PROGRAM Control_LD

VAR	
	Btn1_pressed: BOOL; // Either ixButtLevel1 or ixButtElevat1 was pressed
	Btn2_pressed: BOOL; // Either ixButtLevel2 or ixButtElevat2 was pressed
	Btn3_pressed: BOOL; // Either ixButtLevel3 or ixButtElevat3 was pressed
	Btn_pressed: BOOL; // A button (any button) was pressed
	One_to_two: BOOL; // The command to take the elevator cabin from level 1 to level 2
	One_to_three: BOOL; // The command to take the elevator cabin from level 1 to level 3
	Two_to_three: BOOL; // The command to take the elevator cabin from level 2 to level 3
	Two_to_one: BOOL; // The command to take the elevator cabin from level 2 to level 1
	Three_to_one: BOOL; // The command to take the elevator cabin from level 3 to level 1
	Three_to_two: BOOL; // The command to take the elevator cabin from level 3 to level 2
END_VAR

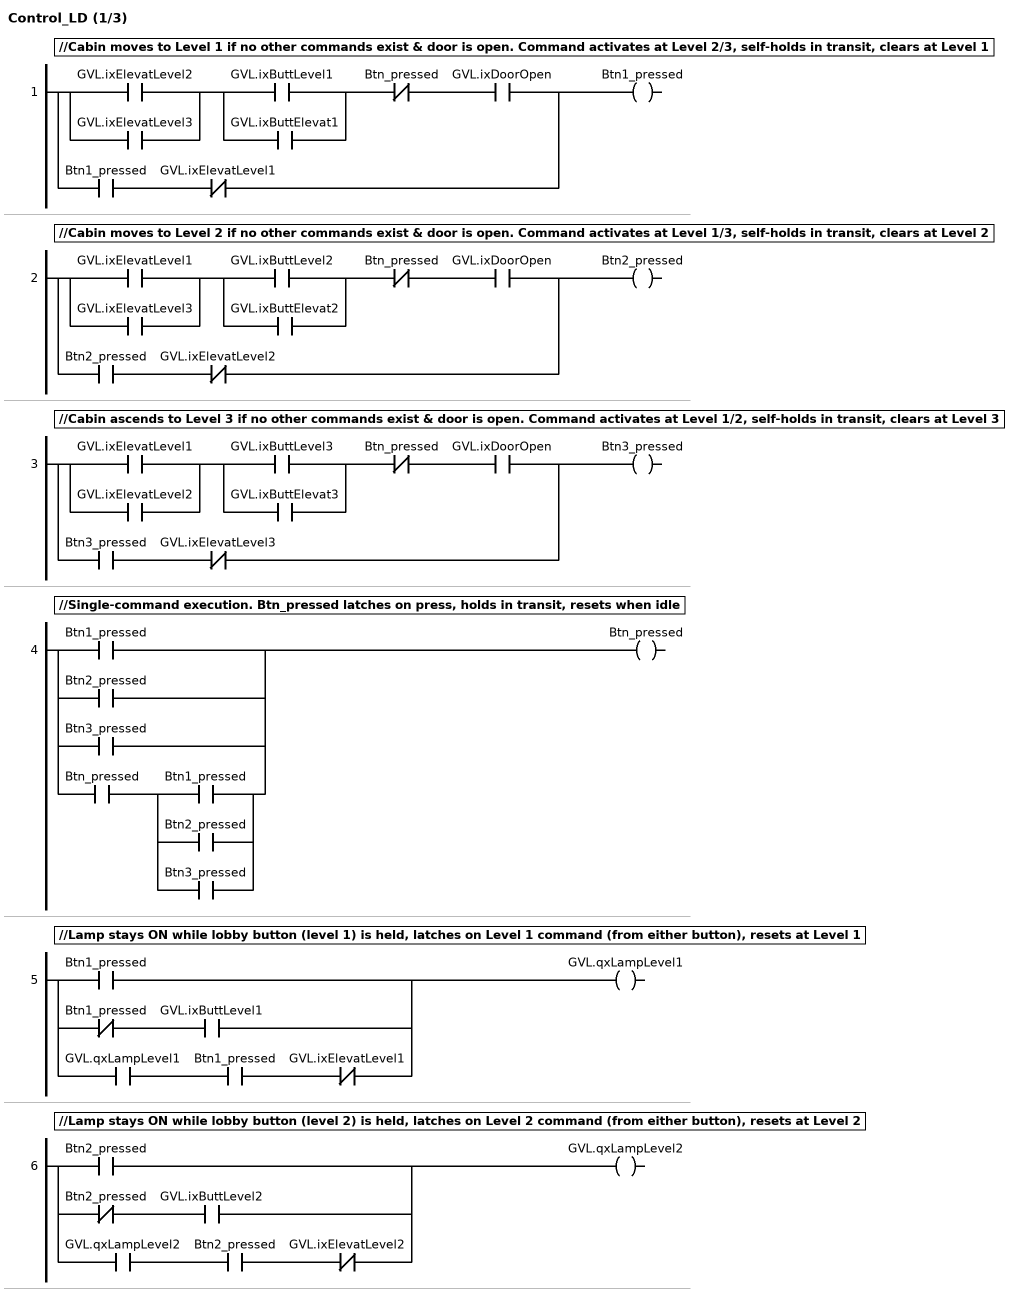
// NETWORK 1
// label: //Cabin moves to Level 1 if no other commands exist & door is open. Command activates at Level 2/3, self-holds in transit, clears at Level 1
Btn1_pressed := (GVL.ixElevatLevel2 OR GVL.ixElevatLevel3) AND (GVL.ixButtLevel1 OR GVL.ixButtElevat1) AND NOT Btn_pressed AND GVL.ixDoorOpen OR Btn1_pressed AND NOT GVL.ixElevatLevel1;

// NETWORK 2
// label: //Cabin moves to Level 2 if no other commands exist & door is open. Command activates at Level 1/3, self-holds in transit, clears at Level 2
Btn2_pressed := (GVL.ixElevatLevel1 OR GVL.ixElevatLevel3) AND (GVL.ixButtLevel2 OR GVL.ixButtElevat2) AND NOT Btn_pressed AND GVL.ixDoorOpen OR Btn2_pressed AND NOT GVL.ixElevatLevel2;

// NETWORK 3
// label: //Cabin ascends to Level 3 if no other commands exist & door is open. Command activates at Level 1/2, self-holds in transit, clears at Level 3
Btn3_pressed := (GVL.ixElevatLevel1 OR GVL.ixElevatLevel2) AND (GVL.ixButtLevel3 OR GVL.ixButtElevat3) AND NOT Btn_pressed AND GVL.ixDoorOpen OR Btn3_pressed AND NOT GVL.ixElevatLevel3;

// NETWORK 4
// label: //Single-command execution. Btn_pressed latches on press, holds in transit, resets when idle
Btn_pressed := Btn1_pressed OR Btn2_pressed OR Btn3_pressed OR Btn_pressed AND (Btn1_pressed OR Btn2_pressed OR Btn3_pressed);

// NETWORK 5
// label: //Lamp stays ON while lobby button (level 1) is held, latches on Level 1 command (from either button), resets at Level 1
GVL.qxLampLevel1 := Btn1_pressed OR NOT Btn1_pressed AND GVL.ixButtLevel1 OR GVL.qxLampLevel1 AND Btn1_pressed AND NOT GVL.ixElevatLevel1;

// NETWORK 6
// label: //Lamp stays ON while lobby button (level 2) is held, latches on Level 2 command (from either button), resets at Level 2
GVL.qxLampLevel2 := Btn2_pressed OR NOT Btn2_pressed AND GVL.ixButtLevel2 OR GVL.qxLampLevel2 AND Btn2_pressed AND NOT GVL.ixElevatLevel2;

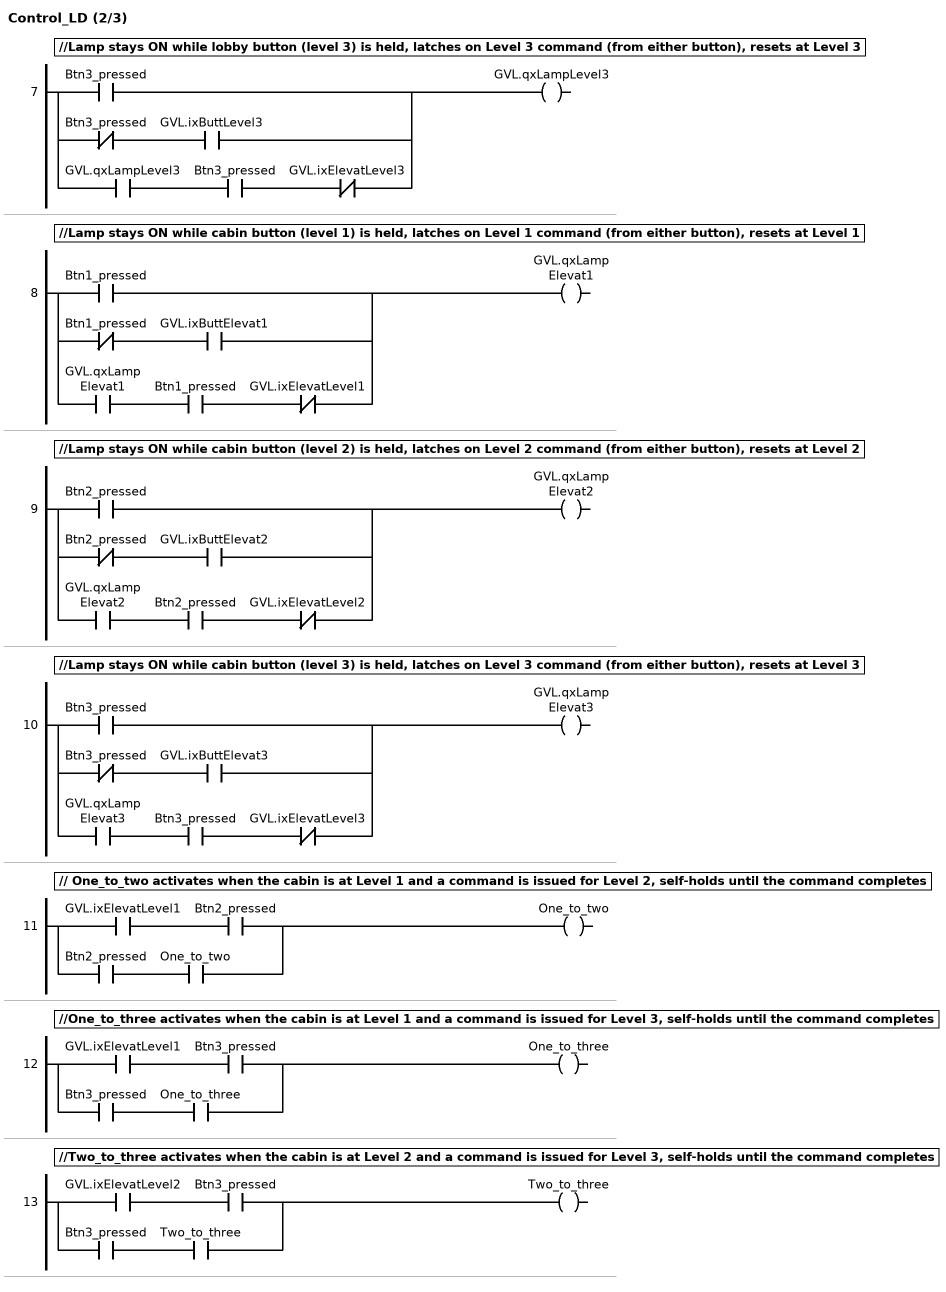
// NETWORK 7
// label: //Lamp stays ON while lobby button (level 3) is held, latches on Level 3 command (from either button), resets at Level 3
GVL.qxLampLevel3 := Btn3_pressed OR NOT Btn3_pressed AND GVL.ixButtLevel3 OR GVL.qxLampLevel3 AND Btn3_pressed AND NOT GVL.ixElevatLevel3;

// NETWORK 8
// label: //Lamp stays ON while cabin button (level 1) is held, latches on Level 1 command (from either button), resets at Level 1
GVL.qxLampElevat1 := Btn1_pressed OR NOT Btn1_pressed AND GVL.ixButtElevat1 OR GVL.qxLampElevat1 AND Btn1_pressed AND NOT GVL.ixElevatLevel1;

// NETWORK 9
// label: //Lamp stays ON while cabin button (level 2) is held, latches on Level 2 command (from either button), resets at Level 2
GVL.qxLampElevat2 := Btn2_pressed OR NOT Btn2_pressed AND GVL.ixButtElevat2 OR GVL.qxLampElevat2 AND Btn2_pressed AND NOT GVL.ixElevatLevel2;

// NETWORK 10
// label: //Lamp stays ON while cabin button (level 3) is held, latches on Level 3 command (from either button), resets at Level 3
GVL.qxLampElevat3 := Btn3_pressed OR NOT Btn3_pressed AND GVL.ixButtElevat3 OR GVL.qxLampElevat3 AND Btn3_pressed AND NOT GVL.ixElevatLevel3;

// NETWORK 11
// label: // One_to_two activates when the cabin is at Level 1 and a command is issued for Level 2, self-holds until the command completes
One_to_two := GVL.ixElevatLevel1 AND Btn2_pressed OR Btn2_pressed AND One_to_two;

// NETWORK 12
// label: //One_to_three activates when the cabin is at Level 1 and a command is issued for Level 3, self-holds until the command completes
One_to_three := GVL.ixElevatLevel1 AND Btn3_pressed OR Btn3_pressed AND One_to_three;

// NETWORK 13
// label: //Two_to_three activates when the cabin is at Level 2 and a command is issued for Level 3, self-holds until the command completes
Two_to_three := GVL.ixElevatLevel2 AND Btn3_pressed OR Btn3_pressed AND Two_to_three;

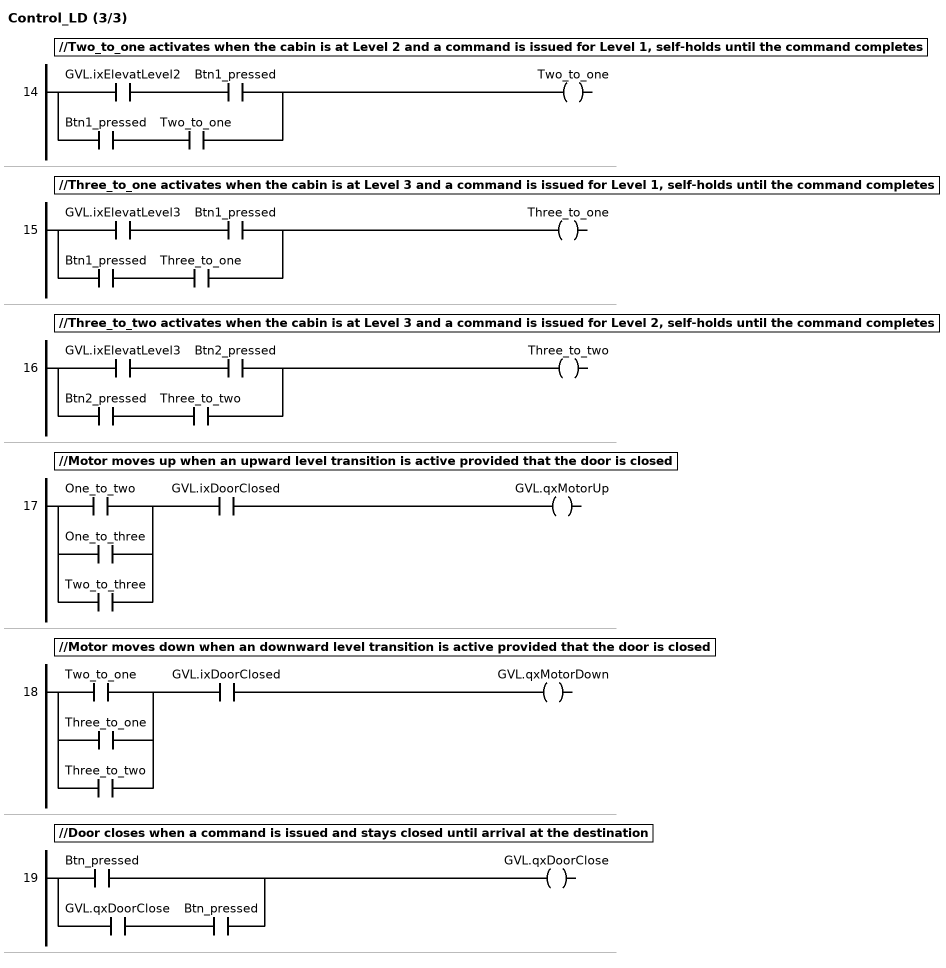
// NETWORK 14
// label: //Two_to_one activates when the cabin is at Level 2 and a command is issued for Level 1, self-holds until the command completes
Two_to_one := GVL.ixElevatLevel2 AND Btn1_pressed OR Btn1_pressed AND Two_to_one;

// NETWORK 15
// label: //Three_to_one activates when the cabin is at Level 3 and a command is issued for Level 1, self-holds until the command completes
Three_to_one := GVL.ixElevatLevel3 AND Btn1_pressed OR Btn1_pressed AND Three_to_one;

// NETWORK 16
// label: //Three_to_two activates when the cabin is at Level 3 and a command is issued for Level 2, self-holds until the command completes
Three_to_two := GVL.ixElevatLevel3 AND Btn2_pressed OR Btn2_pressed AND Three_to_two;

// NETWORK 17
// label: //Motor moves up when an upward level transition is active provided that the door is closed
GVL.qxMotorUp := (One_to_two OR One_to_three OR Two_to_three) AND GVL.ixDoorClosed;

// NETWORK 18
// label: //Motor moves down when an downward level transition is active provided that the door is closed
GVL.qxMotorDown := (Two_to_one OR Three_to_one OR Three_to_two) AND GVL.ixDoorClosed;

// NETWORK 19
// label: //Door closes when a command is issued and stays closed until arrival at the destination
GVL.qxDoorClose := Btn_pressed OR GVL.qxDoorClose AND Btn_pressed;

END_PROGRAM

(* stored: Version 1.1.0.1
   POU Control_LD: Id {912119c4-f197-4ac1-96d5-56b57bc2b241}, SpecialFunc None *)
